// TwinCAT 3 PLC project IO_DigiOut
// Title: IO_DigiOut_Lib
// Company: Chua Siang Poh
// Author: Chua Siang Poh
// ProjectVersion: 1.0
// Description: This library aims to simply reduce the time needed to declare mappable BOOL from the PLC to the IO
// ProgramVersion: 3.1.0.8
// libraries:
//   Tc2_Standard, * (Beckhoff Automation GmbH)
//   Tc2_System, * (Beckhoff Automation GmbH)
//   Tc3_Interfaces, * (Beckhoff Automation GmbH)
//   Tc3_Module, * (Beckhoff Automation GmbH)
// project tree:
//   GVL/ IO_DigiOut_GVL.TcGVL
//   / IO_DigiOut_Parameters.TcGVL
//   Version/ Global_Version.TcGVL

// ---- GVL/IO_DigiOut_GVL.TcGVL
VAR_GLOBAL
	Digital_Output	AT %Q* : ARRAY[1..MAX_D_OUT] OF BOOL;
END_VAR

// ---- IO_DigiOut_Parameters.TcGVL
VAR_GLOBAL CONSTANT
	MAX_D_OUT	: INT := 1;
END_VAR

// ---- Version/Global_Version.TcGVL
// This function has been automatically generated from the project information.
VAR_GLOBAL CONSTANT
	{attribute 'const_non_replaced'}
	stLibVersion_IO_DigiOut_Lib : ST_LibVersion := (iMajor := 1, iMinor := 0, iBuild := 0, iRevision := 0, sVersion := '1.0');
END_VAR
